Staubli VAL3: getFunctionEdit.pgx

public program getFunctionEdit(string& x_sName[])
  local string l_sMessage
begin
  //
  // define your message for the
  // function KEY
  //
  // NOTE is an ARRAY[0..7]
  //
  // example:
  // x_sName[1]="DEMO"
  // active the F2 button
  //
  if (nIndex>0 or jEditPoint.nZoneType==0) and find(jEditPoint.tData[nIndex].tSuper.comment,"@")==-1
    // here
    call language:message(l_sMessage,150)
    x_sName[0]=l_sMessage
  else
  // ALIGN
  call language:message(l_sMessage,134)
  x_sName[1]=l_sMessage
  // Tool
  call language:message(l_sMessage,123)
  x_sName[2]=l_sMessage
  endIf
//  // define the @Link
//  x_sName[1]="@Link"
end
